FUNCTION_BLOCK JSON_PARSER (* Basic FB with empty ECC *)
  (* Standard: 61499-2 *)
  (* Version 1.0, 2023-04-19, valentinnodan *)
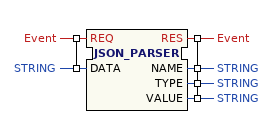
  EVENT_INPUT
    REQ WITH DATA;
  END_EVENT
  EVENT_OUTPUT
    RES WITH NAME, TYPE, VALUE;
  END_EVENT
  VAR_INPUT
    DATA : STRING;
  END_VAR
  VAR_OUTPUT
    NAME : STRING;
    TYPE : STRING;
    VALUE : STRING;
  END_VAR
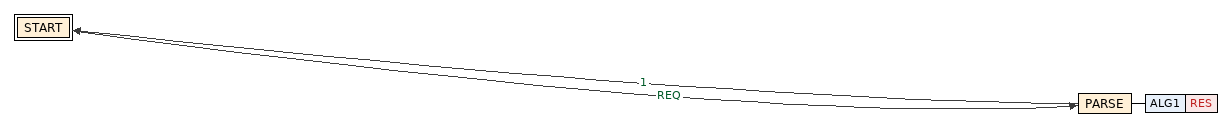
  EC_STATES
    START; (* Initial State *)
    PARSE : ALG1 -> RES;
  END_STATES
  EC_TRANSITIONS
    START TO PARSE := REQ;
    PARSE TO START := 1;
  END_TRANSITIONS
  ALGORITHM ALG1 IN ST:
VAR
     pos : INT;
     currLen: INT;
     inString: BOOL;
     c: STRING;
     fieldType: STRING;
     fieldValue: STRING;
     currField: STRING;
     step: INT;
END_VAR;
step := 1;
WHILE pos < LEN(DATA) DO
    c := MID(DATA, step, pos);
    IF c = '{' THEN (* Start of object *)
        pos := pos + 1;
    ELSIF c = '}' THEN (* End of object *)
    	pos := pos + 1;
    ELSIF c = '"' or c = '$'' THEN (* Start or end of string *)
        IF inString THEN (* End of string *)
            inString := FALSE;
            pos := pos + 1;
        ELSE (* Start of string *)
            inString := TRUE;
            pos := pos + 1;
        END_IF;
    ELSIF c = ':' THEN (* Key-value pair separator *)
        IF NOT inString THEN (* Outside of string *)
            currField := fieldValue;
            fieldValue := "";
            pos := pos + 1;
        ELSE (* Inside of string *)
            fieldValue := CONCAT(fieldValue, c);
            pos := pos + 1;
        END_IF;
    ELSIF c = ',' THEN (* Value separator *)
        IF NOT inString THEN (* Outside of string *)
            IF currField = 'NAME' THEN
                    NAME := fieldValue;
            ELSIF currField = 'TYPE' THEN
                    TYPE :=fieldValue;
             ELSIF currField = 'VALUE' THEN
                    VALUE := fieldValue;
            END_IF;
            currField := '';
            fieldValue := '';
            pos := pos + 1;
        ELSE (* Inside of string *)
            fieldValue := CONCAT(fieldValue, c);
            pos := pos + 1;
        END_IF;
    ELSE (* Other characters *)
        IF inString THEN (* Inside of string *)
            fieldValue := CONCAT(fieldValue, c);
            pos := pos + 1;
        ELSE (* Outside of string *)
            pos := pos + 1;
        END_IF;
    END_IF;
END_WHILE;
IF currField = 'NAME' THEN
        NAME := fieldValue;
ELSIF currField = 'TYPE' THEN
        TYPE :=fieldValue;
 ELSIF currField = 'VALUE' THEN
        VALUE := fieldValue;
END_IF;
  END_ALGORITHM
END_FUNCTION_BLOCK
